FUNCTION_BLOCK FB_Charge
VAR_INPUT
END_VAR
VAR_OUTPUT
END_VAR
VAR
END_VAR

END_FUNCTION_BLOCK

(* stored: Version 1.1.0.1
   POU FB_Charge: Id {28101247-21c0-4e15-930b-d770b5ff78d6}, SpecialFunc None *)
